// TIA Portal V17 export
// export: Created 2023-12-22T15:04:44.7457949Z, ExportSetting WithDefaults, DisplayName Totally Integrated Automation Portal, DisplayVersion V17, DisplayName TIA Portal Openness, DisplayVersion V17, DisplayName TIA Portal Version Control Interface, DisplayVersion V17, DisplayName STEP 7 Professional, DisplayVersion V17, DisplayName STEP 7 Safety, DisplayVersion V17, DisplayName WinCC Advanced, DisplayVersion V17
DATA_BLOCK "ModBus_DB"   // DB20
VERSION : 0.1
// stored: AutoNumber false, DBAccessibleFromOPCUA true, InstanceOfName ModBus, InstanceOfType FB
"ModBus"
   // VAR
   //    "Step" : Int;
   //    "type" : Int;
   //    type_max : Int;
   //    cnt : Int;
   //    cnt_max : Int;
   //    CMD : Struct
   //       DIS : Bool;
   //       REQ : Bool;
   //       BUSY : Bool;
   //       DONE : Bool;
   //       ERROR : Bool;
   //       STATUS : Word;
   //    END_STRUCT;
   //    CFG : Struct
   //       ADDR : UInt;
   //       Register : UDInt;
   //       Length : UInt;
   //       IP : IP_V4;
   //       Port { S7_SetPoint := 'True'} : UInt := 503;
   //       Mode : USInt;
   //    END_STRUCT;
   //    Clock : Array[0..10] of "Time_S";
   //    test : Int;
   //    test_run : Bool;
   // END_VAR
BEGIN
END_DATA_BLOCK
